// TIA Portal project "babu_3WayTrafficInternational_NewWay" (V15)

(* hardware
DEVICE "S7-1200 station_1"  S7-1200 Station
   slot 0: "Rack_0"  S7-1200 Rack  Rack  V1.0
   slot 1: "PLC_1"  CPU 1212C DC/DC/DC  6ES7 212-1AE40-0XB0  V4.2
*)

// ===== PLC "PLC_1"  CPU 1212C DC/DC/DC =====

VAR_GLOBAL   // PLC tag table "Default tag table"
   "POWER BUTTON" AT %I0.0 : Bool;
   "POWER BUTTON MEMORY" AT %M0.1 : Bool;
   "INITIALIZE" AT %M0.2 : Bool;
   "IP2" AT %M0.3 : Bool;
   "OP2" AT %Q0.0 : Bool;
   "IP21" AT %M0.4 : Bool;
   "PP MEMORY" AT %M0.5 : Bool;
   "G3M" AT %M0.6 : Bool;
   "G1M" AT %M0.7 : Bool;
   "G2M" AT %M1.0 : Bool;
   "Y1M" AT %M1.1 : Bool;
   "Y2M" AT %M1.2 : Bool;
   "Y3M" AT %M1.3 : Bool;
   "R1M" AT %M1.4 : Bool;
   "R2M" AT %M1.5 : Bool;
   "R3M" AT %M1.6 : Bool;
   "G1" AT %Q0.1 : Bool;
   "G2" AT %Q0.2 : Bool;
   "G3" AT %Q0.3 : Bool;
   "Y1" AT %Q0.4 : Bool;
   "Y2" AT %Q0.5 : Bool;
   "Y3" AT %Q0.6 : Bool;
   "R1" AT %Q0.7 : Bool;
   "R2" AT %Q1.0 : Bool;
   "R3" AT %Q1.1 : Bool;
   "SEQ1" AT %M0.0 : Bool;
   "SEQ2" AT %M1.7 : Bool;
   "SEQ3" AT %M2.0 : Bool;
   "SEQ4" AT %M2.1 : Bool;
   "SEQ5" AT %M2.2 : Bool;
   "SEQ6" AT %M2.3 : Bool;
   "ERROR" AT %M2.4 : Bool;
   "IP22" AT %M2.5 : Bool;
   "IP22MEM" AT %M2.6 : Bool;
   "OP22" AT %M2.7 : Bool;
   "IP23" AT %M3.0 : Bool;
   "IP24" AT %M3.1 : Bool;
   "IP24MEM" AT %M3.2 : Bool;
   "OP24" AT %Q1.2 : Bool;
   "PP MEM 1" AT %M3.3 : Bool;
   "PP MEM 2" AT %M3.4 : Bool;
   "PP MEM 3" AT %M3.5 : Bool;
   "PP MEM 4" AT %M3.6 : Bool;
   "PP MEM5" AT %M3.7 : Bool;
   "PP MEM6" AT %M4.0 : Bool;
   "PP MEM7" AT %M4.1 : Bool;
   "PP MEM8" AT %M4.2 : Bool;
   "PP MEM9" AT %M4.3 : Bool;
   "SEQ7" AT %M4.4 : Bool;
   "SEQ8" AT %M4.5 : Bool;
   "SEQ9" AT %M4.6 : Bool;
END_VAR

// folder: System blocks/Program resources

DATA_BLOCK "IEC_Timer_0_DB"   // DB1
{ S7_Optimized_Access := 'TRUE' }
AUTHOR : Simatic
FAMILY : IEC
NAME : IEC_TMR
VERSION : 1.0
// stored: InstanceOfName IEC_TIMER
"IEC_TIMER"
BEGIN
END_DATA_BLOCK

DATA_BLOCK "IEC_Timer_0_DB_1"   // DB2
{ S7_Optimized_Access := 'TRUE' }
AUTHOR : Simatic
FAMILY : IEC
NAME : IEC_TMR
VERSION : 1.0
// stored: InstanceOfName IEC_TIMER
"IEC_TIMER"
BEGIN
END_DATA_BLOCK

DATA_BLOCK "IEC_Timer_0_DB_2"   // DB3
{ S7_Optimized_Access := 'TRUE' }
AUTHOR : Simatic
FAMILY : IEC
NAME : IEC_TMR
VERSION : 1.0
// stored: InstanceOfName IEC_TIMER
"IEC_TIMER"
BEGIN
END_DATA_BLOCK

DATA_BLOCK "IEC_Timer_0_DB_3"   // DB4
{ S7_Optimized_Access := 'TRUE' }
AUTHOR : Simatic
FAMILY : IEC
NAME : IEC_TMR
VERSION : 1.0
// stored: InstanceOfName IEC_TIMER
"IEC_TIMER"
BEGIN
END_DATA_BLOCK

DATA_BLOCK "IEC_Timer_0_DB_4"   // DB5
{ S7_Optimized_Access := 'TRUE' }
AUTHOR : Simatic
FAMILY : IEC
NAME : IEC_TMR
VERSION : 1.0
// stored: InstanceOfName IEC_TIMER
"IEC_TIMER"
BEGIN
END_DATA_BLOCK

DATA_BLOCK "IEC_Timer_0_DB_5"   // DB6
{ S7_Optimized_Access := 'TRUE' }
AUTHOR : Simatic
FAMILY : IEC
NAME : IEC_TMR
VERSION : 1.0
// stored: InstanceOfName IEC_TIMER
"IEC_TIMER"
BEGIN
END_DATA_BLOCK

DATA_BLOCK "IEC_Timer_0_DB_6"   // DB7
{ S7_Optimized_Access := 'TRUE' }
AUTHOR : Simatic
FAMILY : IEC
NAME : IEC_TMR
VERSION : 1.0
// stored: InstanceOfName IEC_TIMER
"IEC_TIMER"
BEGIN
END_DATA_BLOCK

DATA_BLOCK "IEC_Timer_0_DB_7"   // DB8
{ S7_Optimized_Access := 'TRUE' }
AUTHOR : Simatic
FAMILY : IEC
NAME : IEC_TMR
VERSION : 1.0
// stored: InstanceOfName IEC_TIMER
"IEC_TIMER"
BEGIN
END_DATA_BLOCK

DATA_BLOCK "IEC_Timer_0_DB_8"   // DB9
{ S7_Optimized_Access := 'TRUE' }
AUTHOR : Simatic
FAMILY : IEC
NAME : IEC_TMR
VERSION : 1.0
// stored: InstanceOfName IEC_TIMER
"IEC_TIMER"
BEGIN
END_DATA_BLOCK

DATA_BLOCK "IEC_Timer_0_DB_11"   // DB12
{ S7_Optimized_Access := 'TRUE' }
AUTHOR : Simatic
FAMILY : IEC
NAME : IEC_TMR
VERSION : 1.0
// stored: InstanceOfName IEC_TIMER
"IEC_TIMER"
BEGIN
END_DATA_BLOCK

DATA_BLOCK "IEC_Timer_0_DB_12"   // DB13
{ S7_Optimized_Access := 'TRUE' }
AUTHOR : Simatic
FAMILY : IEC
NAME : IEC_TMR
VERSION : 1.0
// stored: InstanceOfName IEC_TIMER
"IEC_TIMER"
BEGIN
END_DATA_BLOCK

DATA_BLOCK "IEC_Timer_0_DB_13"   // DB14
{ S7_Optimized_Access := 'TRUE' }
AUTHOR : Simatic
FAMILY : IEC
NAME : IEC_TMR
VERSION : 1.0
// stored: InstanceOfName IEC_TIMER
"IEC_TIMER"
BEGIN
END_DATA_BLOCK

// folder: (top level)

ORGANIZATION_BLOCK "Main"   // OB1, LAD, ProgramCycle
TITLE = "Main Program Sweep (Cycle)"
{ S7_Optimized_Access := 'TRUE' }
VERSION : 0.1
   VAR_INPUT
      Initial_Call : Bool;   // Initial call of this OB
      Remanence : Bool;   // =True, if remanent data are available
   END_VAR
   VAR_TEMP   // added for the SCL form of the ladder/FBD networks
      _w1 : Bool;
      _w2 : Bool;
      _w3 : Bool;
   END_VAR
BEGIN

REGION Network 1: POWER UP
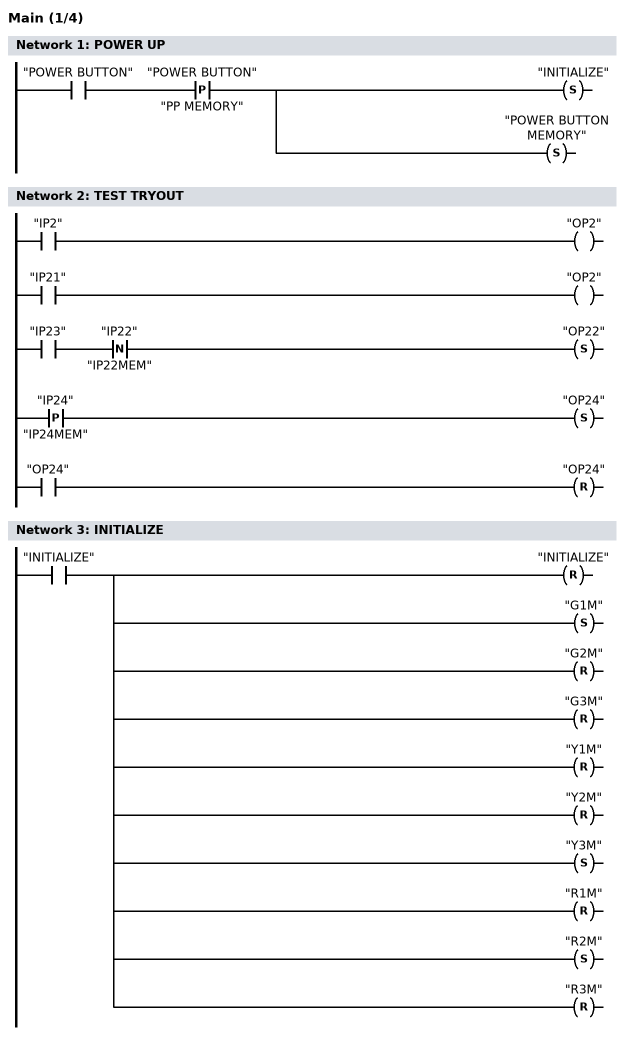
   RUNG wire#powerrail
      Contact( "POWER BUTTON" )
      P_Contact(operand := "POWER BUTTON", bit := "PP MEMORY")
      wire#w1
      S_Coil( "INITIALIZE" )
   END_RUNG
   RUNG wire#w1
      S_Coil( "POWER BUTTON MEMORY" )
   END_RUNG
   // the same network as SCL:
   #_w1 := "POWER BUTTON" AND "POWER BUTTON" AND NOT "PP MEMORY";   // rising edge of "POWER BUTTON"
   "PP MEMORY" := "POWER BUTTON";
   IF #_w1 THEN
       "INITIALIZE" := TRUE;
       "POWER BUTTON MEMORY" := TRUE;
   END_IF;
END_REGION

REGION Network 2: TEST TRYOUT
   RUNG wire#powerrail
      Contact( "IP2" )
      Coil( "OP2" )
   END_RUNG
   RUNG wire#powerrail
      Contact( "IP21" )
      Coil( "OP2" )
   END_RUNG
   RUNG wire#powerrail
      Contact( "IP23" )
      N_Contact(operand := "IP22", bit := "IP22MEM")
      S_Coil( "OP22" )
   END_RUNG
   RUNG wire#powerrail
      P_Contact(operand := "IP24", bit := "IP24MEM")
      S_Coil( "OP24" )
   END_RUNG
   RUNG wire#powerrail
      Contact( "OP24" )
      R_Coil( "OP24" )
   END_RUNG
   // the same network as SCL:
   "OP2" := "IP2";
   "OP2" := "IP21";
   #_w1 := "IP23" AND NOT "IP22" AND "IP22MEM";   // falling edge of "IP22"
   "IP22MEM" := "IP22";
   IF #_w1 THEN "OP22" := TRUE; END_IF;
   #_w2 := "IP24" AND NOT "IP24MEM";   // rising edge of "IP24"
   "IP24MEM" := "IP24";
   IF #_w2 THEN "OP24" := TRUE; END_IF;
   IF "OP24" THEN "OP24" := FALSE; END_IF;
END_REGION

REGION Network 3: INITIALIZE
   RUNG wire#powerrail
      Contact( "INITIALIZE" )
      wire#w1
      R_Coil( "INITIALIZE" )
   END_RUNG
   RUNG wire#w1
      S_Coil( "G1M" )
   END_RUNG
   RUNG wire#w1
      R_Coil( "G2M" )
   END_RUNG
   RUNG wire#w1
      R_Coil( "G3M" )
   END_RUNG
   RUNG wire#w1
      R_Coil( "Y1M" )
   END_RUNG
   RUNG wire#w1
      R_Coil( "Y2M" )
   END_RUNG
   RUNG wire#w1
      S_Coil( "Y3M" )
   END_RUNG
   RUNG wire#w1
      R_Coil( "R1M" )
   END_RUNG
   RUNG wire#w1
      S_Coil( "R2M" )
   END_RUNG
   RUNG wire#w1
      R_Coil( "R3M" )
   END_RUNG
   // the same network as SCL:
   #_w1 := "INITIALIZE";
   IF #_w1 THEN
       "INITIALIZE" := FALSE;
       "G1M" := TRUE;
       "G2M" := FALSE;
       "G3M" := FALSE;
       "Y1M" := FALSE;
       "Y2M" := FALSE;
       "Y3M" := TRUE;
       "R1M" := FALSE;
       "R2M" := TRUE;
       "R3M" := FALSE;
   END_IF;
END_REGION

REGION Network 4: OUTPUT
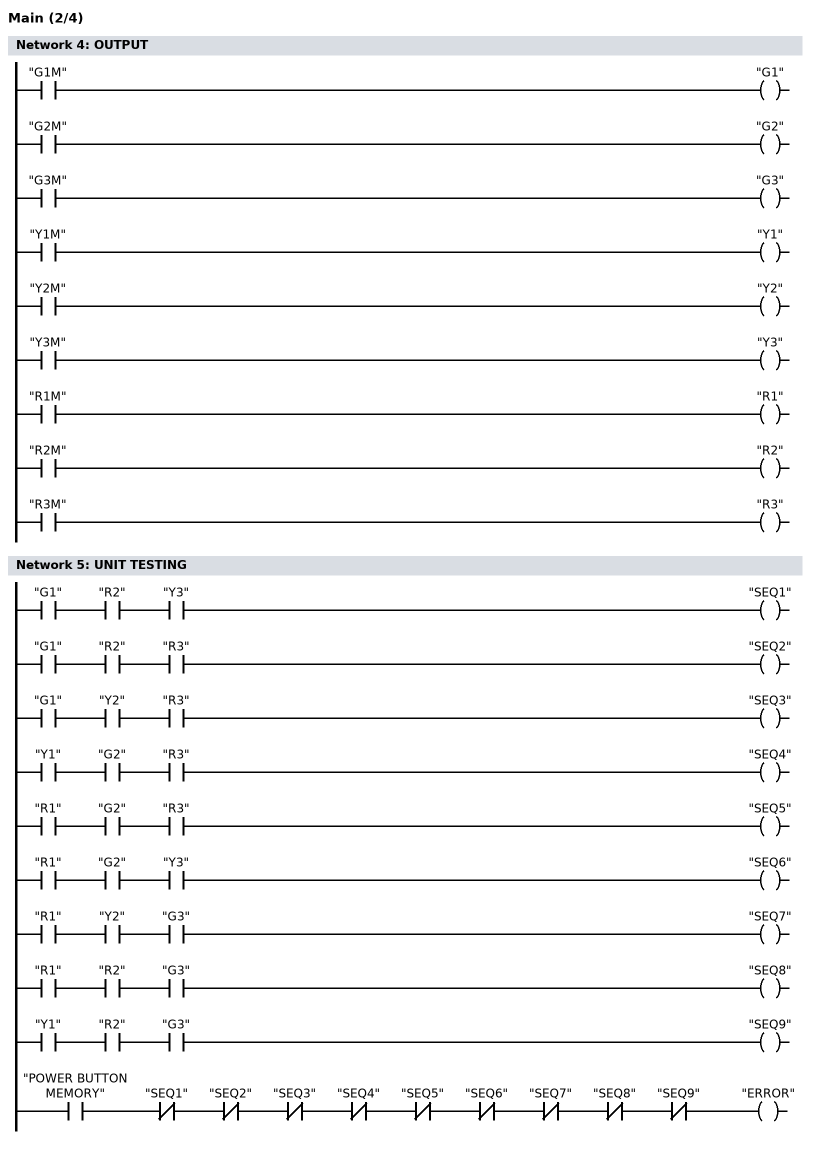
   RUNG wire#powerrail
      Contact( "G1M" )
      Coil( "G1" )
   END_RUNG
   RUNG wire#powerrail
      Contact( "G2M" )
      Coil( "G2" )
   END_RUNG
   RUNG wire#powerrail
      Contact( "G3M" )
      Coil( "G3" )
   END_RUNG
   RUNG wire#powerrail
      Contact( "Y1M" )
      Coil( "Y1" )
   END_RUNG
   RUNG wire#powerrail
      Contact( "Y2M" )
      Coil( "Y2" )
   END_RUNG
   RUNG wire#powerrail
      Contact( "Y3M" )
      Coil( "Y3" )
   END_RUNG
   RUNG wire#powerrail
      Contact( "R1M" )
      Coil( "R1" )
   END_RUNG
   RUNG wire#powerrail
      Contact( "R2M" )
      Coil( "R2" )
   END_RUNG
   RUNG wire#powerrail
      Contact( "R3M" )
      Coil( "R3" )
   END_RUNG
   // the same network as SCL:
   "G1" := "G1M";
   "G2" := "G2M";
   "G3" := "G3M";
   "Y1" := "Y1M";
   "Y2" := "Y2M";
   "Y3" := "Y3M";
   "R1" := "R1M";
   "R2" := "R2M";
   "R3" := "R3M";
END_REGION

REGION Network 5: UNIT TESTING
   RUNG wire#powerrail
      Contact( "G1" )
      Contact( "R2" )
      Contact( "Y3" )
      Coil( "SEQ1" )
   END_RUNG
   RUNG wire#powerrail
      Contact( "G1" )
      Contact( "R2" )
      Contact( "R3" )
      Coil( "SEQ2" )
   END_RUNG
   RUNG wire#powerrail
      Contact( "G1" )
      Contact( "Y2" )
      Contact( "R3" )
      Coil( "SEQ3" )
   END_RUNG
   RUNG wire#powerrail
      Contact( "Y1" )
      Contact( "G2" )
      Contact( "R3" )
      Coil( "SEQ4" )
   END_RUNG
   RUNG wire#powerrail
      Contact( "R1" )
      Contact( "G2" )
      Contact( "R3" )
      Coil( "SEQ5" )
   END_RUNG
   RUNG wire#powerrail
      Contact( "R1" )
      Contact( "G2" )
      Contact( "Y3" )
      Coil( "SEQ6" )
   END_RUNG
   RUNG wire#powerrail
      Contact( "R1" )
      Contact( "Y2" )
      Contact( "G3" )
      Coil( "SEQ7" )
   END_RUNG
   RUNG wire#powerrail
      Contact( "R1" )
      Contact( "R2" )
      Contact( "G3" )
      Coil( "SEQ8" )
   END_RUNG
   RUNG wire#powerrail
      Contact( "Y1" )
      Contact( "R2" )
      Contact( "G3" )
      Coil( "SEQ9" )
   END_RUNG
   RUNG wire#powerrail
      Contact( "POWER BUTTON MEMORY" )
      I_Contact( "SEQ1" )
      I_Contact( "SEQ2" )
      I_Contact( "SEQ3" )
      I_Contact( "SEQ4" )
      I_Contact( "SEQ5" )
      I_Contact( "SEQ6" )
      I_Contact( "SEQ7" )
      I_Contact( "SEQ8" )
      I_Contact( "SEQ9" )
      Coil( "ERROR" )
   END_RUNG
   // the same network as SCL:
   "SEQ1" := "G1" AND "R2" AND "Y3";
   "SEQ2" := "G1" AND "R2" AND "R3";
   "SEQ3" := "G1" AND "Y2" AND "R3";
   "SEQ4" := "Y1" AND "G2" AND "R3";
   "SEQ5" := "R1" AND "G2" AND "R3";
   "SEQ6" := "R1" AND "G2" AND "Y3";
   "SEQ7" := "R1" AND "Y2" AND "G3";
   "SEQ8" := "R1" AND "R2" AND "G3";
   "SEQ9" := "Y1" AND "R2" AND "G3";
   "ERROR" := "POWER BUTTON MEMORY" AND NOT "SEQ1" AND NOT "SEQ2" AND NOT "SEQ3" AND NOT "SEQ4" AND NOT "SEQ5" AND NOT "SEQ6" AND NOT "SEQ7" AND NOT "SEQ8" AND NOT "SEQ9";
END_REGION

REGION Network 6: G3
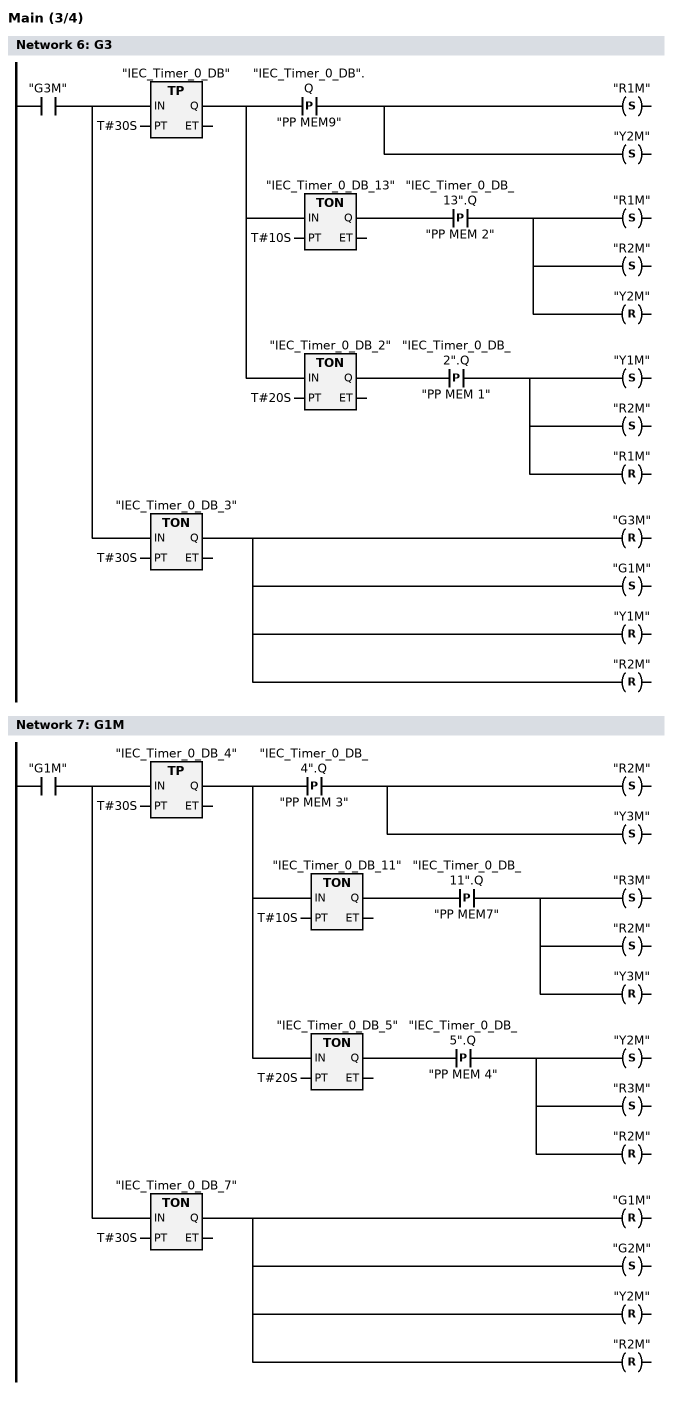
   "IEC_Timer_0_DB".TP(IN := "G3M", PT := T#30S);
   #_w1 := "IEC_Timer_0_DB".Q AND "IEC_Timer_0_DB".Q AND NOT "PP MEM9";   // rising edge of "IEC_Timer_0_DB".Q
   "PP MEM9" := "IEC_Timer_0_DB".Q;
   IF #_w1 THEN
       "R1M" := TRUE;
       "Y2M" := TRUE;
   END_IF;
   "IEC_Timer_0_DB_13".TON(IN := "IEC_Timer_0_DB".Q, PT := T#10S);
   #_w2 := "IEC_Timer_0_DB_13".Q AND "IEC_Timer_0_DB_13".Q AND NOT "PP MEM 2";   // rising edge of "IEC_Timer_0_DB_13".Q
   "PP MEM 2" := "IEC_Timer_0_DB_13".Q;
   IF #_w2 THEN
       "R1M" := TRUE;
       "R2M" := TRUE;
       "Y2M" := FALSE;
   END_IF;
   "IEC_Timer_0_DB_2".TON(IN := "IEC_Timer_0_DB".Q, PT := T#20S);
   #_w3 := "IEC_Timer_0_DB_2".Q AND "IEC_Timer_0_DB_2".Q AND NOT "PP MEM 1";   // rising edge of "IEC_Timer_0_DB_2".Q
   "PP MEM 1" := "IEC_Timer_0_DB_2".Q;
   IF #_w3 THEN
       "Y1M" := TRUE;
       "R2M" := TRUE;
       "R1M" := FALSE;
   END_IF;
   "IEC_Timer_0_DB_3".TON(IN := "G3M", PT := T#30S);
   IF "IEC_Timer_0_DB_3".Q THEN
       "G3M" := FALSE;
       "G1M" := TRUE;
       "Y1M" := FALSE;
       "R2M" := FALSE;
   END_IF;
END_REGION

REGION Network 7: G1M
   "IEC_Timer_0_DB_4".TP(IN := "G1M", PT := T#30S);
   #_w1 := "IEC_Timer_0_DB_4".Q AND "IEC_Timer_0_DB_4".Q AND NOT "PP MEM 3";   // rising edge of "IEC_Timer_0_DB_4".Q
   "PP MEM 3" := "IEC_Timer_0_DB_4".Q;
   IF #_w1 THEN
       "R2M" := TRUE;
       "Y3M" := TRUE;
   END_IF;
   "IEC_Timer_0_DB_11".TON(IN := "IEC_Timer_0_DB_4".Q, PT := T#10S);
   #_w2 := "IEC_Timer_0_DB_11".Q AND "IEC_Timer_0_DB_11".Q AND NOT "PP MEM7";   // rising edge of "IEC_Timer_0_DB_11".Q
   "PP MEM7" := "IEC_Timer_0_DB_11".Q;
   IF #_w2 THEN
       "R3M" := TRUE;
       "R2M" := TRUE;
       "Y3M" := FALSE;
   END_IF;
   "IEC_Timer_0_DB_5".TON(IN := "IEC_Timer_0_DB_4".Q, PT := T#20S);
   #_w3 := "IEC_Timer_0_DB_5".Q AND "IEC_Timer_0_DB_5".Q AND NOT "PP MEM 4";   // rising edge of "IEC_Timer_0_DB_5".Q
   "PP MEM 4" := "IEC_Timer_0_DB_5".Q;
   IF #_w3 THEN
       "Y2M" := TRUE;
       "R3M" := TRUE;
       "R2M" := FALSE;
   END_IF;
   "IEC_Timer_0_DB_7".TON(IN := "G1M", PT := T#30S);
   IF "IEC_Timer_0_DB_7".Q THEN
       "G1M" := FALSE;
       "G2M" := TRUE;
       "Y2M" := FALSE;
       "R2M" := FALSE;
   END_IF;
END_REGION

REGION Network 8: G2
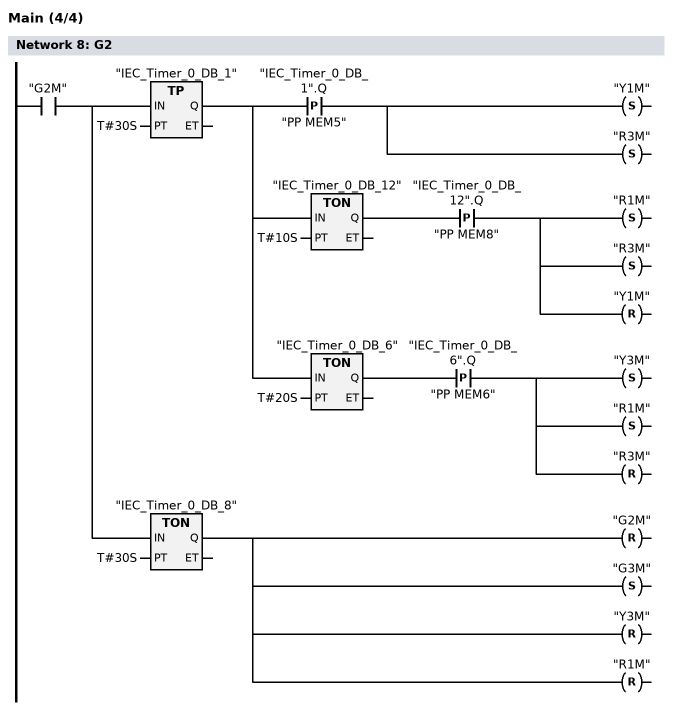
   "IEC_Timer_0_DB_1".TP(IN := "G2M", PT := T#30S);
   #_w1 := "IEC_Timer_0_DB_1".Q AND "IEC_Timer_0_DB_1".Q AND NOT "PP MEM5";   // rising edge of "IEC_Timer_0_DB_1".Q
   "PP MEM5" := "IEC_Timer_0_DB_1".Q;
   IF #_w1 THEN
       "Y1M" := TRUE;
       "R3M" := TRUE;
   END_IF;
   "IEC_Timer_0_DB_12".TON(IN := "IEC_Timer_0_DB_1".Q, PT := T#10S);
   #_w2 := "IEC_Timer_0_DB_12".Q AND "IEC_Timer_0_DB_12".Q AND NOT "PP MEM8";   // rising edge of "IEC_Timer_0_DB_12".Q
   "PP MEM8" := "IEC_Timer_0_DB_12".Q;
   IF #_w2 THEN
       "R1M" := TRUE;
       "R3M" := TRUE;
       "Y1M" := FALSE;
   END_IF;
   "IEC_Timer_0_DB_6".TON(IN := "IEC_Timer_0_DB_1".Q, PT := T#20S);
   #_w3 := "IEC_Timer_0_DB_6".Q AND "IEC_Timer_0_DB_6".Q AND NOT "PP MEM6";   // rising edge of "IEC_Timer_0_DB_6".Q
   "PP MEM6" := "IEC_Timer_0_DB_6".Q;
   IF #_w3 THEN
       "Y3M" := TRUE;
       "R1M" := TRUE;
       "R3M" := FALSE;
   END_IF;
   "IEC_Timer_0_DB_8".TON(IN := "G2M", PT := T#30S);
   IF "IEC_Timer_0_DB_8".Q THEN
       "G2M" := FALSE;
       "G3M" := TRUE;
       "Y3M" := FALSE;
       "R1M" := FALSE;
   END_IF;
END_REGION
END_ORGANIZATION_BLOCK